// TIA Portal V20 export
DATA_BLOCK "InterfaceTP_C4"   // DB411
// stored: Access Published, MemoryReserve 100, Namespace Conveyor4
   VAR
      operationOFF : Bool;   // operation ON (HMI) manual mode
      operationON : Bool;   // operation ON (HMI) automatic mode
      jogRight : Bool;   // jog conveyor right
      jogLeft : Bool;   // jog conveyor left
      acknowledgeFault : Bool;   // acknowledge conveyor fault
      actualValue : UInt;   // actual value
      setpoint : UInt := 3;   // setpoint value
      operation : Bool;
      conveyorFault : Bool;
   END_VAR
BEGIN
END_DATA_BLOCK
